TYPE
    ST_DualChannel_HMIStatus : STRUCT
		Name : STRING;
		Status_Usint : USINT;
		Status_Str : STRING;		
    END_STRUCT
END_TYPE

(* stored: Version 1.1.0.1
   DUT ST_DualChannel_HMIStatus: Id {271a1248-9541-4000-9842-7b2ce5624e1b} *)
